FUNCTION_BLOCK ABSTRACT VisionNode EXTENDS Node IMPLEMENTS I_PreCheckedNode
VAR
	preExecutionCheckExtension : PreExecutionCheckExtension('precheck', THIS^);
	watchdogCheckExtension : WatchdogCheckExtension('watchdog', THIS^);
END_VAR

METHOD PUBLIC Execute
VAR
END_VAR
IF NOT preExecutionCheckExtension.Check() THEN
	RETURN;
END_IF

watchdogCheckExtension.Start();
SUPER^.Execute();
watchdogCheckExtension.Stop();
END_METHOD

METHOD PUBLIC ABSTRACT PreExecutionCheck
VAR_INPUT
	Check : I_PreExecutionChecks;
END_VAR
END_METHOD

END_FUNCTION_BLOCK

(* stored: Version 1.1.0.1, ProductVersion 3.1.4026.18
   POU VisionNode: Id {f924a3b9-a7ea-048f-393e-cff5c17d2882}, SpecialFunc None
   Method Execute: Id {8505f98d-9e97-07b5-148b-0e469a2003d1}
   Method PreExecutionCheck: Id {1cc0fb1a-9fc7-05d0-0dda-466734a3a96c} *)
